TYPE ST_MqttData :
STRUCT
	
	stTopic					: STRING(255);
	stMessage				: STRING(255);

END_STRUCT
END_TYPE

(* stored: Version 1.1.0.1, ProductVersion 3.1.4024.12
   DUT ST_MqttData: Id {dd86d567-b8b1-4f2f-bb61-09888b2151f7} *)
